(* CoDeSys 2.3 export: ERR_RESET.EXP *)

(* POU Alarm/ERR_RESET, ST *)
FUNCTION ERR_RESET : BOOL
VAR_INPUT
	Num: INT; (* Номер ошибки *)
END_VAR
VAR
END_VAR
	glbErrors[Num].LatchState := glbErrors[Num].State := FALSE;
END_FUNCTION
